Yaskawa INFORM job: kufsa_angle.JBI

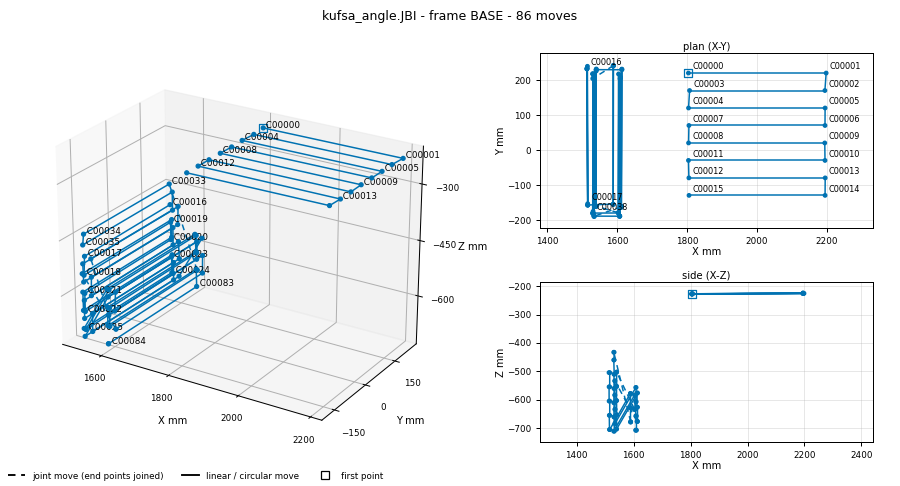
[picture p0: tool path of kufsa_angle.JBI in frame BASE, 86 of 91 moves have a stored position in this frame; points joined in program order, loops and branches not executed]
/JOB
//NAME kufsa_angle
//POS
///NPOS 86,0,86,0,0,0
///TOOL 0
///POSTYPE BASE
///RECTAN
///RCONF 0,0,0,0,0,0,0,0,0,0,0,0,0,0,0,0,0,0,0,0,0,0,0,0
C00000=1804.266325,220.599653,-227.332738,179.000000,1.000000,1.000000
C00001=2198.370318,220.599653,-225.837376,179.000000,1.000000,1.000000
C00002=2194.801646,170.599653,-225.649258,179.000000,1.000000,1.000000
C00003=1807.577372,170.599653,-227.559024,179.000000,1.000000,1.000000
C00004=1804.622430,120.599653,-227.769031,179.000000,1.000000,1.000000
C00005=2195.335932,120.599653,-225.843218,179.000000,1.000000,1.000000
C00006=2195.106227,70.599653,-225.320928,179.000000,1.000000,1.000000
C00007=1805.716129,70.599653,-228.029358,179.000000,1.000000,1.000000
C00008=1804.735379,20.599653,-228.045950,179.000000,1.000000,1.000000
C00009=2194.418889,20.599653,-225.391268,179.000000,1.000000,1.000000
C00010=2195.097343,-29.400347,-225.681507,179.000000,1.000000,1.000000
C00011=1804.440697,-29.400347,-228.141761,179.000000,1.000000,1.000000
C00012=1805.619171,-79.400347,-227.256088,179.000000,1.000000,1.000000
C00013=2195.630614,-79.400347,-225.700903,179.000000,1.000000,1.000000
C00014=2195.292275,-129.400347,-224.241996,179.000000,1.000000,1.000000
C00015=1805.953195,-129.400347,-227.208183,179.000000,1.000000,1.000000
C00016=1513.631371,232.354105,-503.993759,179.000000,-89.999999,1.000000
C00017=1516.149493,-153.231824,-503.993759,179.000000,-89.999999,1.000000
C00018=1516.042636,-157.471041,-553.993759,179.000000,-89.999999,1.000000
C00019=1513.923007,233.133060,-553.993759,179.000000,-89.999999,1.000000
C00020=1514.033164,233.523618,-603.993759,179.000000,-89.999999,1.000000
C00021=1516.196196,-156.884002,-603.993759,179.000000,-89.999999,1.000000
C00022=1516.145432,-156.999537,-653.993759,179.000000,-89.999999,1.000000
C00023=1514.649686,233.710250,-653.993759,179.000000,-89.999999,1.000000
C00024=1515.282961,239.938289,-703.993759,179.000000,-89.999999,1.000000
C00025=1516.324119,-157.007223,-703.993759,179.000000,-89.999999,1.000000
C00026=1588.761352,-154.348255,-577.217063,180.000000,-45.000000,0.000000
C00027=1588.933694,240.643984,-577.217063,180.000000,-45.000000,0.000000
C00028=1588.993849,242.129355,-627.217063,180.000000,-45.000000,0.000000
C00029=1589.153246,-155.140421,-627.217063,180.000000,-45.000000,0.000000
C00030=1589.056288,-155.290063,-677.217063,180.000000,-45.000000,0.000000
C00031=1589.812156,241.960017,-677.217063,180.000000,-45.000000,0.000000
C00032=1589.812156,241.960017,-677.217063,180.000000,-45.000000,0.000000
C00033=1530.443677,204.779526,-432.522984,179.000000,-89.999999,1.000000
C00034=1531.499338,-175.214887,-432.522984,179.000000,-89.999999,1.000000
C00035=1531.405902,-179.918631,-459.727325,179.000000,-89.999999,1.000000
C00036=1530.485711,218.119278,-459.727325,179.000000,-89.999999,1.000000
C00037=1531.882210,216.269711,-509.727325,179.000000,-89.999999,1.000000
C00038=1531.275956,-181.949677,-509.727325,179.000000,-89.999999,1.000000
C00039=1531.305500,-180.389462,-559.727325,179.000000,-89.999999,1.000000
C00040=1531.688372,217.320008,-559.727325,179.000000,-89.999999,1.000000
C00041=1530.439594,218.736562,-609.727325,179.000000,-89.999999,1.000000
C00042=1531.606946,-180.718155,-609.727325,179.000000,-89.999999,1.000000
C00043=1530.852010,-180.562819,-659.727325,179.000000,-89.999999,1.000000
C00044=1531.645377,217.737283,-659.727325,179.000000,-89.999999,1.000000
C00045=1532.334739,216.222247,-709.727325,179.000000,-89.999999,1.000000
C00046=1530.209246,-180.083358,-709.727325,179.000000,-89.999999,1.000000
C00047=1603.447683,-179.797306,-582.950629,180.000000,-45.000000,0.000000
C00048=1605.418250,217.726115,-582.950629,180.000000,-45.000000,0.000000
C00049=1604.594618,217.605806,-632.950629,180.000000,-45.000000,0.000000
C00050=1603.382590,-179.006665,-632.950629,180.000000,-45.000000,0.000000
C00051=1603.382590,-179.006665,-632.950629,180.000000,-45.000000,0.000000
C00052=1540.494889,-160.372879,-502.282786,179.000000,-89.999999,1.000000
C00053=1540.352752,230.020570,-502.282786,179.000000,-89.999999,1.000000
C00054=1540.533216,226.582647,-552.282786,179.000000,-89.999999,1.000000
C00055=1540.232062,-160.082242,-552.282786,179.000000,-89.999999,1.000000
C00056=1539.904510,-161.733829,-602.282786,179.000000,-89.999999,1.000000
C00057=1540.218482,229.622326,-602.282786,179.000000,-89.999999,1.000000
C00058=1540.573319,232.252230,-652.282786,179.000000,-89.999999,1.000000
C00059=1540.340568,-160.160305,-652.282786,179.000000,-89.999999,1.000000
C00060=1539.291795,-159.918188,-702.282786,179.000000,-89.999999,1.000000
C00061=1540.509611,230.302320,-702.282786,179.000000,-89.999999,1.000000
C00062=1613.808299,230.041227,-575.506091,180.000000,-45.000000,0.000000
C00063=1612.459514,-160.195374,-575.506091,180.000000,-45.000000,0.000000
C00064=1611.652882,-164.339713,-625.506091,180.000000,-45.000000,0.000000
C00065=1613.824290,231.968799,-625.506091,180.000000,-45.000000,0.000000
C00066=1613.735454,230.903530,-675.506091,180.000000,-45.000000,0.000000
C00067=1612.429310,-162.123426,-675.506091,180.000000,-45.000000,0.000000
C00068=1612.429310,-162.123426,-675.506091,180.000000,-45.000000,0.000000
C00069=1534.042848,-189.208300,-533.001296,179.000000,-89.999999,1.000000
C00070=1534.110824,208.321467,-533.001296,179.000000,-89.999999,1.000000
C00071=1533.962863,207.490215,-583.001296,179.000000,-89.999999,1.000000
C00072=1534.342373,-189.439527,-583.001296,179.000000,-89.999999,1.000000
C00073=1534.609951,-189.394094,-633.001296,179.000000,-89.999999,1.000000
C00074=1534.722122,207.440213,-633.001296,179.000000,-89.999999,1.000000
C00075=1535.013960,204.575123,-683.001296,179.000000,-89.999999,1.000000
C00076=1534.488412,-188.796354,-683.001296,179.000000,-89.999999,1.000000
C00077=1607.894986,-189.015652,-556.224601,180.000000,-45.000000,0.000000
C00078=1608.406843,204.586037,-556.224601,180.000000,-45.000000,0.000000
C00079=1609.291244,208.155978,-606.224601,180.000000,-45.000000,0.000000
C00080=1607.577927,-189.129362,-606.224601,180.000000,-45.000000,0.000000
C00081=1607.618040,-188.869707,-656.224601,180.000000,-45.000000,0.000000
C00082=1609.664028,207.585650,-656.224601,180.000000,-45.000000,0.000000
C00083=1610.137454,208.269434,-706.224601,180.000000,-45.000000,0.000000
C00084=1607.691780,-188.817929,-706.224601,180.000000,-45.000000,0.000000
C00085=1607.691780,-188.817929,-706.224601,180.000000,-45.000000,0.000000
///POSTYPE PULSE
///PULSE
EC00000=0
EC00001=0
EC00002=0
EC00003=0
EC00004=0
EC00005=0
EC00006=0
EC00007=0
EC00008=0
EC00009=0
EC00010=0
EC00011=0
EC00012=0
EC00013=0
EC00014=0
EC00015=0
EC00016=0
EC00017=0
EC00018=0
EC00019=0
EC00020=0
EC00021=0
EC00022=0
EC00023=0
EC00024=0
EC00025=0
EC00026=0
EC00027=0
EC00028=0
EC00029=0
EC00030=0
EC00031=0
EC00032=92160
EC00033=92160
EC00034=92160
EC00035=92160
EC00036=92160
EC00037=92160
EC00038=92160
EC00039=92160
EC00040=92160
EC00041=92160
EC00042=92160
EC00043=92160
EC00044=92160
EC00045=92160
EC00046=92160
EC00047=92160
EC00048=92160
EC00049=92160
EC00050=92160
EC00051=184320
EC00052=184320
EC00053=184320
EC00054=184320
EC00055=184320
EC00056=184320
EC00057=184320
EC00058=184320
EC00059=184320
EC00060=184320
EC00061=184320
EC00062=184320
EC00063=184320
EC00064=184320
EC00065=184320
EC00066=184320
EC00067=184320
EC00068=276480
EC00069=276480
EC00070=276480
EC00071=276480
EC00072=276480
EC00073=276480
EC00074=276480
EC00075=276480
EC00076=276480
EC00077=276480
EC00078=276480
EC00079=276480
EC00080=276480
EC00081=276480
EC00082=276480
EC00083=276480
EC00084=276480
EC00085=368640
//INST
///DATE 2023/01/18 16:57
///ATTR SC,RW,RJ
////FRAME BASE
///GROUP1 RB1,ST1
NOP
MOVJ C00000 EC00000 VJ=15.0
SPYON
MOVL C00001 EC00001 V=200.0
MOVL C00002 EC00002 V=200.0
MOVL C00003 EC00003 V=200.0
MOVL C00004 EC00004 V=200.0
MOVL C00005 EC00005 V=200.0
MOVL C00006 EC00006 V=200.0
MOVL C00007 EC00007 V=200.0
MOVL C00008 EC00008 V=200.0
MOVL C00009 EC00009 V=200.0
MOVL C00010 EC00010 V=200.0
MOVL C00011 EC00011 V=200.0
MOVL C00012 EC00012 V=200.0
MOVL C00013 EC00013 V=200.0
MOVL C00014 EC00014 V=200.0
MOVL C00015 EC00015 V=200.0
SPYOF
MOVJ P009 VJ=15.00
MOVJ C00016 EC00016 VJ=15.0
SPYON
MOVL C00017 EC00017 V=200.0
MOVL C00018 EC00018 V=200.0
MOVL C00019 EC00019 V=200.0
MOVL C00020 EC00020 V=200.0
MOVL C00021 EC00021 V=200.0
MOVL C00022 EC00022 V=200.0
MOVL C00023 EC00023 V=200.0
MOVL C00024 EC00024 V=200.0
MOVL C00025 EC00025 V=200.0
MOVL C00026 EC00026 V=200.0
MOVL C00027 EC00027 V=200.0
MOVL C00028 EC00028 V=200.0
MOVL C00029 EC00029 V=200.0
MOVL C00030 EC00030 V=200.0
MOVL C00031 EC00031 V=200.0
SPYOF
MOVJ P009 VJ=15.00
MOVL C00032 EC00032 V=200.0
MOVJ C00033 EC00033 VJ=15.0
SPYON
MOVL C00034 EC00034 V=200.0
MOVL C00035 EC00035 V=200.0
MOVL C00036 EC00036 V=200.0
MOVL C00037 EC00037 V=200.0
MOVL C00038 EC00038 V=200.0
MOVL C00039 EC00039 V=200.0
MOVL C00040 EC00040 V=200.0
MOVL C00041 EC00041 V=200.0
MOVL C00042 EC00042 V=200.0
MOVL C00043 EC00043 V=200.0
MOVL C00044 EC00044 V=200.0
MOVL C00045 EC00045 V=200.0
MOVL C00046 EC00046 V=200.0
MOVL C00047 EC00047 V=200.0
MOVL C00048 EC00048 V=200.0
MOVL C00049 EC00049 V=200.0
MOVL C00050 EC00050 V=200.0
SPYOF
MOVJ P009 VJ=15.00
MOVL C00051 EC00051 V=200.0
MOVJ C00052 EC00052 VJ=15.0
SPYON
MOVL C00053 EC00053 V=200.0
MOVL C00054 EC00054 V=200.0
MOVL C00055 EC00055 V=200.0
MOVL C00056 EC00056 V=200.0
MOVL C00057 EC00057 V=200.0
MOVL C00058 EC00058 V=200.0
MOVL C00059 EC00059 V=200.0
MOVL C00060 EC00060 V=200.0
MOVL C00061 EC00061 V=200.0
MOVL C00062 EC00062 V=200.0
MOVL C00063 EC00063 V=200.0
MOVL C00064 EC00064 V=200.0
MOVL C00065 EC00065 V=200.0
MOVL C00066 EC00066 V=200.0
MOVL C00067 EC00067 V=200.0
SPYOF
MOVJ P009 VJ=15.00
MOVL C00068 EC00068 V=200.0
MOVJ C00069 EC00069 VJ=15.0
SPYON
MOVL C00070 EC00070 V=200.0
MOVL C00071 EC00071 V=200.0
MOVL C00072 EC00072 V=200.0
MOVL C00073 EC00073 V=200.0
MOVL C00074 EC00074 V=200.0
MOVL C00075 EC00075 V=200.0
MOVL C00076 EC00076 V=200.0
MOVL C00077 EC00077 V=200.0
MOVL C00078 EC00078 V=200.0
MOVL C00079 EC00079 V=200.0
MOVL C00080 EC00080 V=200.0
MOVL C00081 EC00081 V=200.0
MOVL C00082 EC00082 V=200.0
MOVL C00083 EC00083 V=200.0
MOVL C00084 EC00084 V=200.0
SPYOF
MOVJ P009 VJ=15.00
MOVL C00085 EC00085 V=200.0
END
